SUBAPPLICATION Ventilsteuerung_Uebung_020g (* DigitalInput_I1 auf DigitalOutput_Q1; E_TONOF; Ein-/Ausschaltverzögert *)
  (* Standard: 61499-2 *)
  (* Version 1.0, 2023-10-23, franz *)
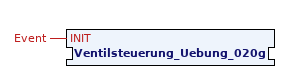
  EVENT_INPUT
    INIT;
  END_EVENT
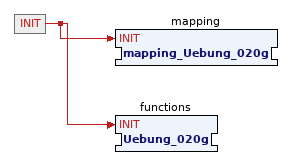
  SUBAPPS
    mapping : mapping_Uebung_020g;
    functions : Uebung_020g;
  END_SUBAPPS
  EVENT_CONNECTIONS
    INIT TO mapping.INIT;
    INIT TO functions.INIT;
  END_CONNECTIONS
END_SUBAPPLICATION
